TYPE eMainState :
(
	init		:= 0,
	ready		:= 10,
	output		:= 20,
	separation	:= 30,
	refill		:= 40,
	emergencyStop	:= 50,
	error			:= 60,
	resetSystem		:= 70
);
END_TYPE

(* stored: Version 1.1.0.1, ProductVersion 3.1.0.25
   DUT eMainState: Id {78593579-3f95-451d-9ae5-bf03315db0c9} *)
